// LS Electric XG5000 project: 반입_코드
// PLC LSPLC

PROGRAM NewProgram (task: 스캔 프로그램)

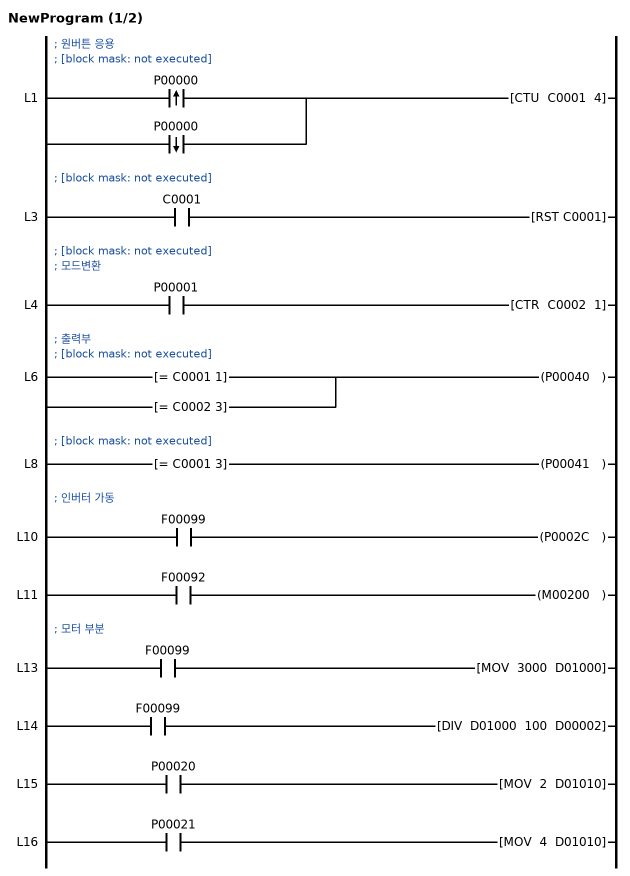
// 원버튼 응용
; L1 (block mask: not executed)
LOADP     P00000
ORN       P00000
CTU       C0001 4
; L3 (block mask: not executed)
LOAD      C0001
RST       C0001
; L4 (block mask: not executed)
LOAD      P00001
CTR       C0002 1
// output comment: 모드변환
// 출력부
; L6 (block mask: not executed)
LOAD=     C0001 1
OR=       C0002 3
OUT       P00040
; L8 (block mask: not executed)
LOAD=     C0001 3
OUT       P00041
// 인버터 가동
; L10
LOAD      F00099
OUT       P0002C
; L11
LOAD      F00092
OUT       M00200
// 모터 부분
; L13
LOAD      F00099
MOV       3000 D01000
; L14
LOAD      F00099
DIV       D01000 100 D00002
; L15
LOAD      P00020
MOV       2 D01010
; L16
LOAD      P00021
MOV       4 D01010

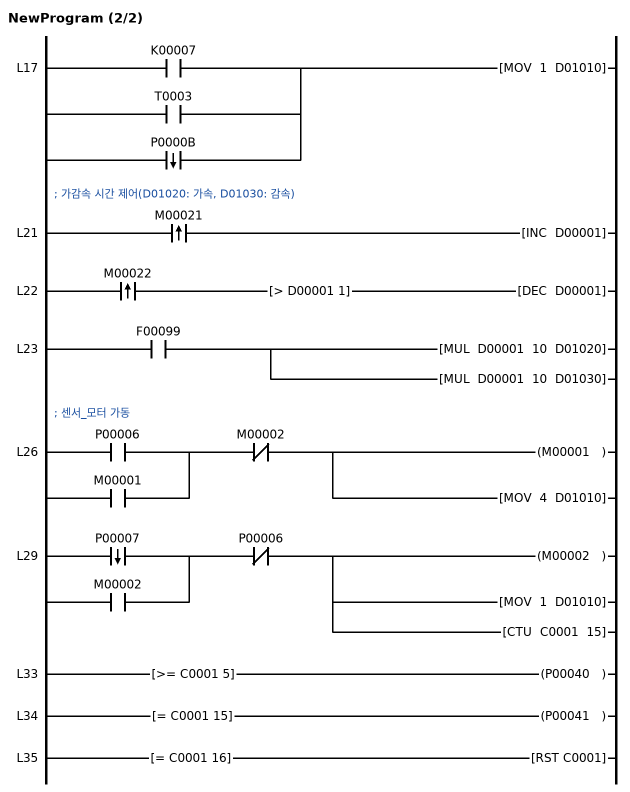
; L17
LOAD      K00007
OR        T0003
ORN       P0000B
MOV       1 D01010
// 가감속 시간 제어(D01020: 가속, D01030: 감속)
; L21
LOADP     M00021
INC       D00001
; L22
LOADP     M00022
AND>      D00001 1
DEC       D00001
; L23
LOAD      F00099
MUL       D00001 10 D01020
MUL       D00001 10 D01030
// 센서_모터 가동
; L26
LOAD      P00006
OR        M00001
AND NOT   M00002
OUT       M00001
MOV       4 D01010
; L29
LOADN     P00007
OR        M00002
AND NOT   P00006
OUT       M00002
MOV       1 D01010
CTU       C0001 15
; L33
LOAD>=    C0001 5
OUT       P00040
; L34
LOAD=     C0001 15
OUT       P00041
; L35
LOAD=     C0001 16
RST       C0001